(* Logix 5000 project; controller CarbonScout_MK6 vendor 1 type 14 code 154 rev 32.11; software revision 32.00; part 11 of 17 *)
(* tags used below, declared in another part *)
   ManualRunning : BOOL;
   ONS : BOOL[32];
   AI_FIT_01 : P_AIn;   // Purge water flow
   AI_LIT_01 : P_AIn;   // Carbon Scout Laser Level Transmitter
   AI_LIT_02 : P_AIn;   // Carbon Scout Cone Level Transmitter
   AI_PIT_01 : P_AIn;   // Water supply pressure
   AI_WIT_01 : P_AIn;   // Weight measure
   CS_Alarms : P_Alarm[80];
   CS_DINTParams : DINT[100];
   CS_REALParams : REAL[80];   // CS REAL Parameters
   CS_Result : CS_Results;   // Sample Result Live Async
   CS_Seq : GEK_Sequence;
   CS_Seq_ControlStop : BOOL;
   CS_Seq_CrashStop : BOOL;
   CS_Tank : CS_TankParams[20];
   CS_Timer : TIMER[80];
   CS_XRF : XRF;
   FOQ02 : TOTALIZER;   // Radar Calibration Totaliser
   N51 : DINT[5];   // From Client
   Oneshot : DINT;
   Oneshot2 : DINT;
   Oneshot3 : DINT;
   TimeAndDate : DINT[7];
   Valve_XV_01 : P_ValveSO;   // Sample Valve Tank 1
   Valve_XV_02 : P_ValveSO;   // Sample Valve Tank 2
   Valve_XV_03 : P_ValveSO;   // Sample Valve Tank 3
   Valve_XV_04 : P_ValveSO;   // Sample Valve Tank 4
   Valve_XV_05 : P_ValveSO;   // Sample Valve Tank 5
   Valve_XV_06 : P_ValveSO;   // Sample Valve Tank 6
   Valve_XV_07 : P_ValveSO;   // Sample Valve Tank 7
   Valve_XV_08 : P_ValveSO;   // Sample Valve Tank 8
   Valve_XV_09 : P_ValveSO;   // Sample Valve Tank 9
   Valve_XV_10 : P_ValveSO;   // Sample Valve Tank 10
   Valve_XV_11 : P_ValveSO;   // Purge Valve
   Valve_XV_12 : P_ValveSO;   // Slurry inlet vavle
   Valve_XV_13 : P_ValveSO;   // Sample line vavle
   Valve_XV_14 : P_ValveSO;   // Top wash vavle
   Valve_XV_15 : P_ValveSO;   // Bottme wash vavle
   Valve_XV_16 : P_ValveSO;   // Potable water valve / Supply Water Valve
   Valve_XV_17 : P_ValveSO;   // Sample cone outlet vavle
   Valve_XV_18 : P_ValveSO;   // Sample strainer discharge
   Valve_XV_19 : P_ValveSO;   // Laser window
(* SeqProgram, continued *)

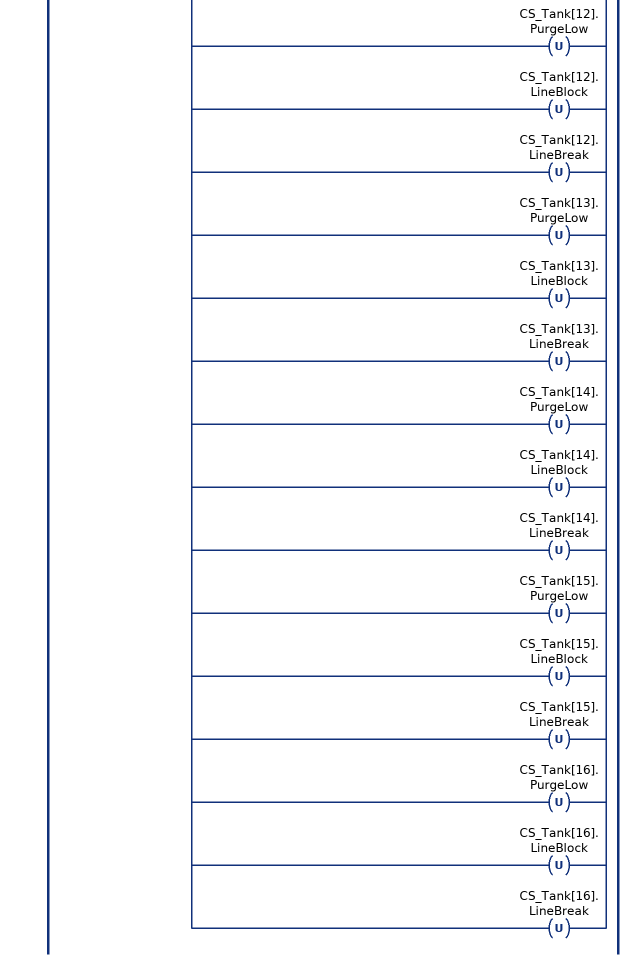
   83: XIC(CS_Seq.HMI_Reset_Req)[OTU(CS_Tank[1].PurgeLow) ,OTU(CS_Tank[1].LineBlock) ,OTU(CS_Tank[1].LineBreak) ,OTU(CS_Tank[2].PurgeLow) ,OTU(CS_Tank[2].LineBlock) ,OTU(CS_Tank[2].LineBreak) ,OTU(CS_Tank[3].PurgeLow) ,OTU(CS_Tank[3].LineBlock) ,OTU(CS_Tank[3].LineBreak) ,OTU(CS_Tank[4].PurgeLow) ,OTU(CS_Tank[4].LineBlock) ,OTU(CS_Tank[4].LineBreak) ,OTU(CS_Tank[5].PurgeLow) ,OTU(CS_Tank[5].LineBlock) ,OTU(CS_Tank[5].LineBreak) ,OTU(CS_Tank[6].PurgeLow) ,OTU(CS_Tank[6].LineBlock) ,OTU(CS_Tank[6].LineBreak) ,OTU(CS_Tank[7].PurgeLow) ,OTU(CS_Tank[7].LineBlock) ,OTU(CS_Tank[7].LineBreak) ,OTU(CS_Tank[8].PurgeLow) ,OTU(CS_Tank[8].LineBlock) ,OTU(CS_Tank[8].LineBreak) ,OTU(CS_Tank[9].PurgeLow) ,OTU(CS_Tank[9].LineBlock) ,OTU(CS_Tank[9].LineBreak) ,OTU(CS_Tank[10].PurgeLow) ,OTU(CS_Tank[10].LineBlock) ,OTU(CS_Tank[10].LineBreak) ,OTU(CS_Tank[11].PurgeLow) ,OTU(CS_Tank[11].LineBlock) ,OTU(CS_Tank[11].LineBreak) ,OTU(CS_Tank[12].PurgeLow) ,OTU(CS_Tank[12].LineBlock) ,OTU(CS_Tank[12].LineBreak) ,OTU(CS_Tank[13].PurgeLow) ,OTU(CS_Tank[13].LineBlock) ,OTU(CS_Tank[13].LineBreak) ,OTU(CS_Tank[14].PurgeLow) ,OTU(CS_Tank[14].LineBlock) ,OTU(CS_Tank[14].LineBreak) ,OTU(CS_Tank[15].PurgeLow) ,OTU(CS_Tank[15].LineBlock) ,OTU(CS_Tank[15].LineBreak) ,OTU(CS_Tank[16].PurgeLow) ,OTU(CS_Tank[16].LineBlock) ,OTU(CS_Tank[16].LineBreak) ];
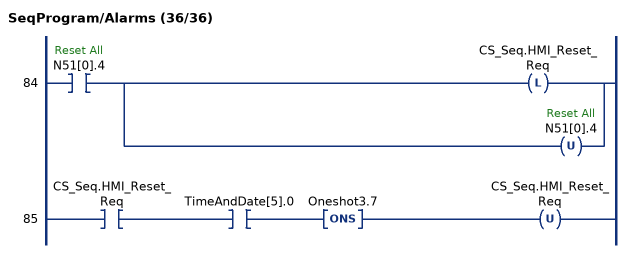
   84: XIC(N51[0].4)[OTL(CS_Seq.HMI_Reset_Req) ,OTU(N51[0].4) ];
   85: XIC(CS_Seq.HMI_Reset_Req)XIC(TimeAndDate[5].0)ONS(Oneshot3.7)OTU(CS_Seq.HMI_Reset_Req);
END_ROUTINE

ROUTINE AutoControl   (* ladder *)
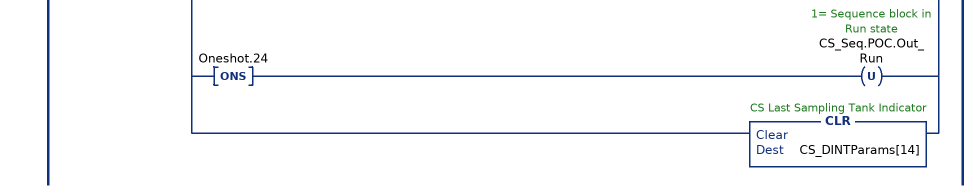
   // +++++++++++++++++++++++++++++
   // Gekko Batch/Continous Sequencer
   // Developed by TL and BT
   // +++++++++++++++++++++++++++++
   0: [MOV(0,CS_DINTParams[0]) P_Mode(CS_Seq.Mode) ,OTL(CS_Seq.Mode.Cfg_ProgDefault) ,DIV(CS_Seq.SeqTimer[0].ACC,1000,CS_DINTParams[1]) ,[XIC(CS_Seq.Mode.Sts_Prog) [[XIC(CS_Seq.HMI_Start_Req) ,XIC(CS_Timer[78].DN) ,XIC(N51[0].5) XIC(N51[0].0) ,XIC(CS_Seq.POC.Sts_Stopped) XIC(CS_DINTParams[99].11) [XIC(CS_DINTParams[97].0) XIC(CS_DINTParams[97].10) ,XIC(CS_DINTParams[97].1) XIC(CS_DINTParams[97].11) ,XIC(CS_DINTParams[97].2) XIC(CS_DINTParams[97].12) ,XIC(CS_DINTParams[97].3) XIC(CS_DINTParams[97].13) ,XIC(CS_DINTParams[97].4) XIC(CS_DINTParams[97].14) ,XIC(CS_DINTParams[97].5) XIC(CS_DINTParams[97].15) ,XIC(CS_DINTParams[97].6) XIC(CS_DINTParams[97].16) ,XIC(CS_DINTParams[97].7) XIC(CS_DINTParams[97].17) ,XIC(CS_DINTParams[97].8) XIC(CS_DINTParams[97].18) ,XIC(CS_DINTParams[97].9) XIC(CS_DINTParams[97].19) ] ] OTE(CS_Seq.POC.In_Cmd_Start) ,[XIC(CS_Seq.HMI_Pause_Req) ,LIM(1,N51[2],10) ] OTE(CS_Seq.POC.In_Cmd_Pause) ,[XIC(CS_Seq.HMI_StopPause_Req) ,XIC(N51[0].5) XIC(N51[0].1) ,LIM(11,N51[2],20) ] [AFI() OTE(CS_Seq.POC.In_Cmd_StopPause) ,OTL(CS_Seq_ControlStop) ] ] ,XIC(CS_Seq.Mode.Sts_Prog) [XIC(CS_Seq.HMI_Resume_Req) ,XIC(CS_Timer[78].DN) ] OTE(CS_Seq.POC.In_Cmd_Resume) ,XIC(CS_Seq.HMI_SkipF_Req) OTE(CS_Seq.POC.In_Cmd_SkipF) ,XIC(CS_Seq.HMI_SkipR_Req) OTE(CS_Seq.POC.In_Cmd_SkipR) ] ,OTL(CS_Seq.POC.In_Cfg_BatchContinous) MOV(23,CS_Seq.POC.In_MaxStepNum) MOV(2147483647,CS_Seq.SeqTimer[0].PRE) GekkoSeq(CS_Seq.POC,CS_Seq.SeqTimer[0]) ,[XIC(CS_Seq.POC.Sts_Running) ,XIC(CS_Seq.POC.Out_Run) ] [ONS(Oneshot.21) MOV(CS_Seq.POC.Out_MovingStepNum,CS_Seq.ActiveStage) ,MOV(CS_Seq.ActiveStage,CS_Seq.POC.In_StepNum) MOV(CS_Seq.ActiveStage,CS_Seq.POC.Out_MovingStepNum) ] ,XIC(CS_Seq.POC.Sts_Resumed) MOV(CS_Seq.POC.Out_NewStepNum,CS_Seq.ActiveStage) ,[XIO(CS_Seq.POC.Out_Run) XIO(CS_Seq.POC.Sts_StopPaused) XIO(CS_Seq.POC.Sts_Paused) XIO(CS_Seq.POC.Sts_Resumed) ,[[[XIC(CS_Seq_CrashStop) ,LIM(21,N51[2],30) ] ,XIC(S:FS) ] [CLR(CS_DINTParams[39]) ,OTU(CS_DINTParams[98].10) ] ,XIC(CS_Alarms[2].Alm) ] CLR(CS_Seq.POC.Out_MovingStepNum) ] MOV(0,CS_Seq.ActiveStage) ,EQU(CS_Seq.ActiveStage,0) OTE(CS_Seq.POC.In_Stopped) ,XIC(CS_Seq.POC.Out_Run) NEQ(CS_Seq.ActiveStage,0) OTE(CS_Seq.POC.In_Running) ,XIC(CS_Seq.POC.Sts_Stopped) [XIC(CS_Seq.POC.Sts_Paused) OTU(CS_Seq.POC.Sts_Paused) ,XIC(CS_Seq.POC.Sts_StopPaused) OTU(CS_Seq.POC.Sts_StopPaused) ,OTU(CS_Seq_ControlStop) ,OTU(CS_DINTParams[99].23) ,OTU(CS_DINTParams[99].10) ,OTU(CS_DINTParams[99].7) MOV(0,CS_Result.ErrorFlag) ,OTU(CS_DINTParams[99].8) ,ONS(Oneshot.24) OTU(CS_Seq.POC.Out_Run) ,CLR(CS_DINTParams[14]) ] ];
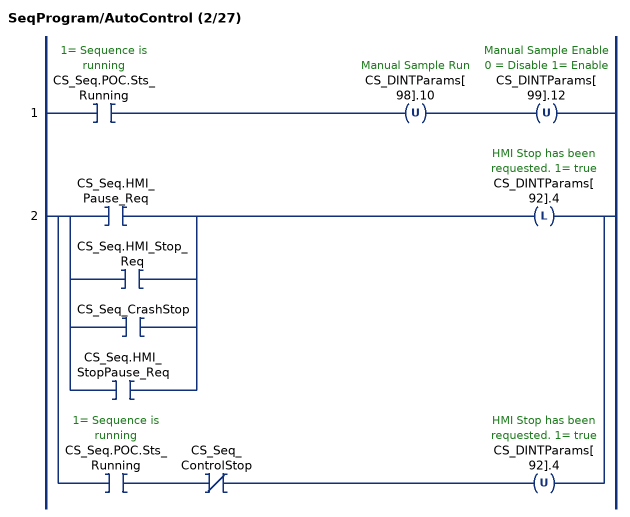
   1: XIC(CS_Seq.POC.Sts_Running)OTU(CS_DINTParams[98].10)OTU(CS_DINTParams[99].12);
   2: [[XIC(CS_Seq.HMI_Pause_Req) ,XIC(CS_Seq.HMI_Stop_Req) ,XIC(CS_Seq_CrashStop) ,XIC(CS_Seq.HMI_StopPause_Req) ] OTL(CS_DINTParams[92].4) ,XIC(CS_Seq.POC.Sts_Running) XIO(CS_Seq_ControlStop) OTU(CS_DINTParams[92].4) ];
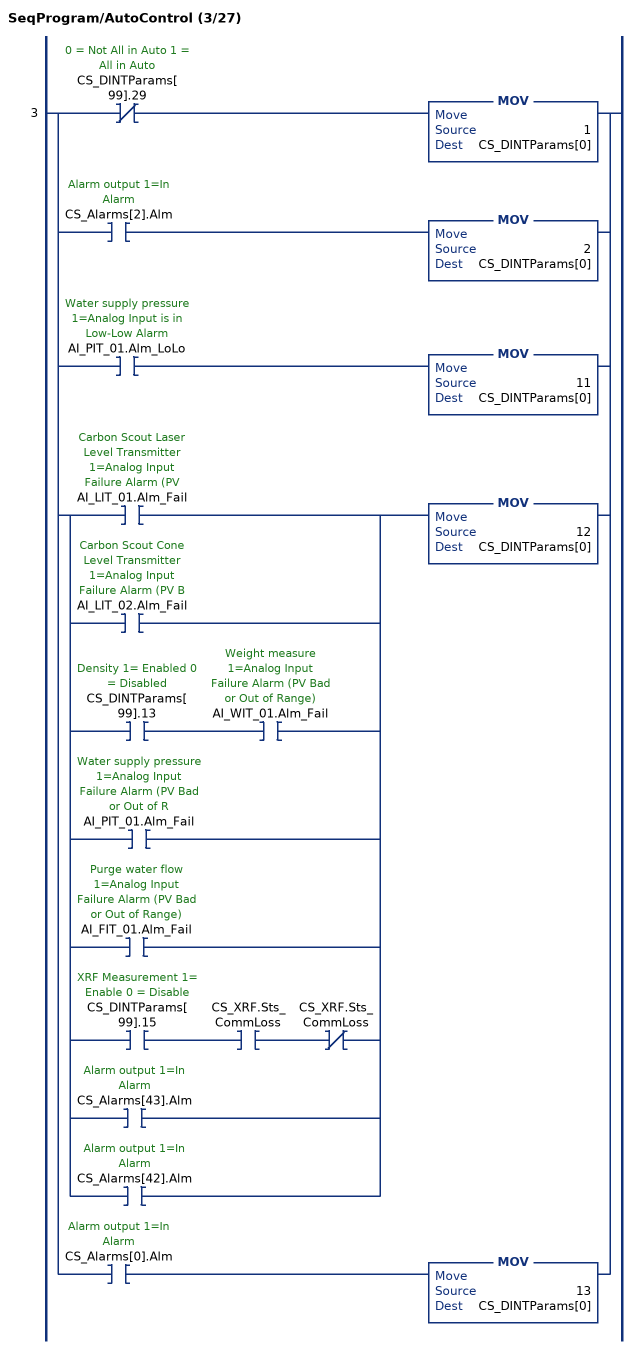
   3: [XIO(CS_DINTParams[99].29) MOV(1,CS_DINTParams[0]) ,XIC(CS_Alarms[2].Alm) MOV(2,CS_DINTParams[0]) ,XIC(AI_PIT_01.Alm_LoLo) MOV(11,CS_DINTParams[0]) ,[XIC(AI_LIT_01.Alm_Fail) ,XIC(AI_LIT_02.Alm_Fail) ,XIC(CS_DINTParams[99].13) XIC(AI_WIT_01.Alm_Fail) ,XIC(AI_PIT_01.Alm_Fail) ,XIC(AI_FIT_01.Alm_Fail) ,XIC(CS_DINTParams[99].15) XIC(CS_XRF.Sts_CommLoss) XIO(CS_XRF.Sts_CommLoss) ,XIC(CS_Alarms[43].Alm) ,XIC(CS_Alarms[42].Alm) ] MOV(12,CS_DINTParams[0]) ,XIC(CS_Alarms[0].Alm) MOV(13,CS_DINTParams[0]) ];
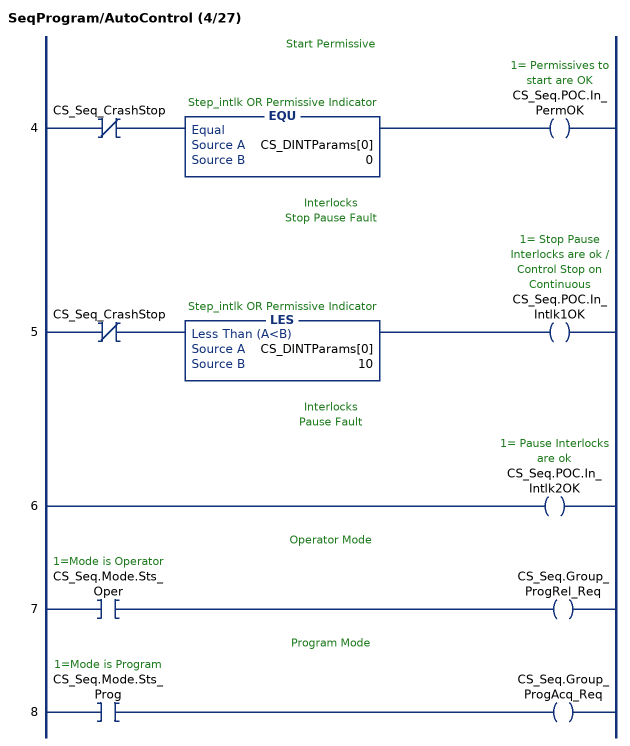
   // Start Permissive
   4: XIO(CS_Seq_CrashStop)EQU(CS_DINTParams[0],0)OTE(CS_Seq.POC.In_PermOK);
   // Interlocks
   // Stop Pause Fault
   5: XIO(CS_Seq_CrashStop)LES(CS_DINTParams[0],10)OTE(CS_Seq.POC.In_Intlk1OK);
   // Interlocks
   // Pause Fault
   6: OTE(CS_Seq.POC.In_Intlk2OK);
   // Operator Mode
   7: XIC(CS_Seq.Mode.Sts_Oper)OTE(CS_Seq.Group_ProgRel_Req);
   // Program Mode
   8: XIC(CS_Seq.Mode.Sts_Prog)OTE(CS_Seq.Group_ProgAcq_Req);
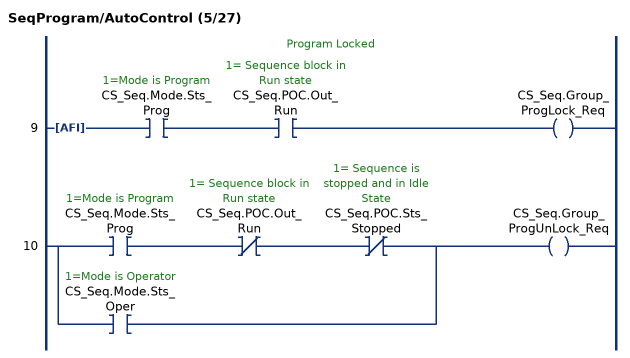
   // Program Locked
   9: AFI()XIC(CS_Seq.Mode.Sts_Prog)XIC(CS_Seq.POC.Out_Run)OTE(CS_Seq.Group_ProgLock_Req);
   10: [XIC(CS_Seq.Mode.Sts_Prog) XIO(CS_Seq.POC.Out_Run) XIO(CS_Seq.POC.Sts_Stopped) ,XIC(CS_Seq.Mode.Sts_Oper) ]OTE(CS_Seq.Group_ProgUnLock_Req);
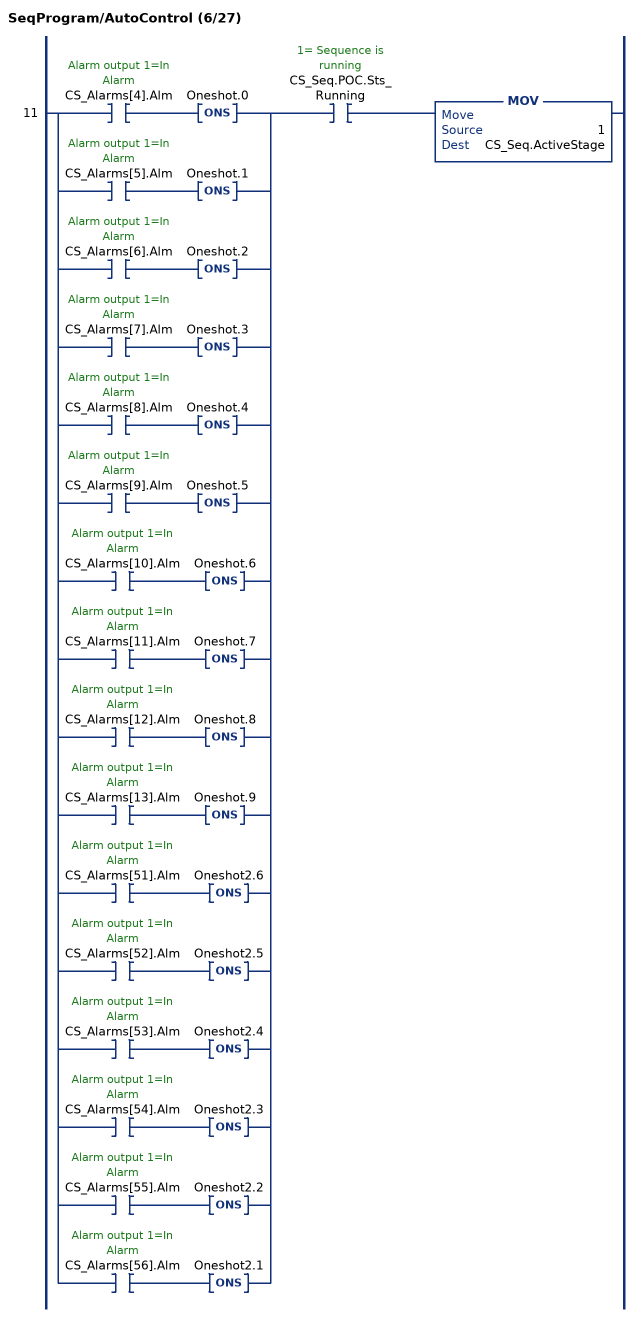
   11: [XIC(CS_Alarms[4].Alm) ONS(Oneshot.0) ,XIC(CS_Alarms[5].Alm) ONS(Oneshot.1) ,XIC(CS_Alarms[6].Alm) ONS(Oneshot.2) ,XIC(CS_Alarms[7].Alm) ONS(Oneshot.3) ,XIC(CS_Alarms[8].Alm) ONS(Oneshot.4) ,XIC(CS_Alarms[9].Alm) ONS(Oneshot.5) ,XIC(CS_Alarms[10].Alm) ONS(Oneshot.6) ,XIC(CS_Alarms[11].Alm) ONS(Oneshot.7) ,XIC(CS_Alarms[12].Alm) ONS(Oneshot.8) ,XIC(CS_Alarms[13].Alm) ONS(Oneshot.9) ,XIC(CS_Alarms[51].Alm) ONS(Oneshot2.6) ,XIC(CS_Alarms[52].Alm) ONS(Oneshot2.5) ,XIC(CS_Alarms[53].Alm) ONS(Oneshot2.4) ,XIC(CS_Alarms[54].Alm) ONS(Oneshot2.3) ,XIC(CS_Alarms[55].Alm) ONS(Oneshot2.2) ,XIC(CS_Alarms[56].Alm) ONS(Oneshot2.1) ]XIC(CS_Seq.POC.Sts_Running)MOV(1,CS_Seq.ActiveStage);
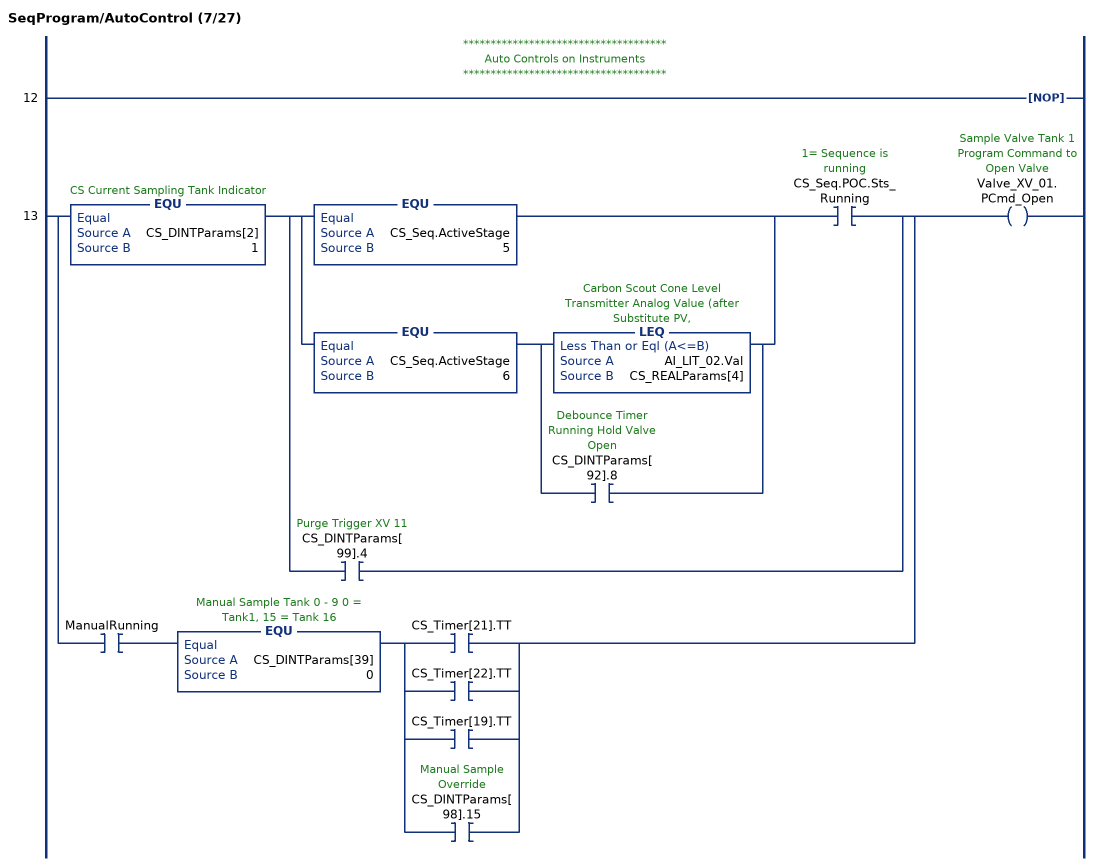
   // *************************************
   // Auto Controls on Instruments
   // *************************************
   12: NOP();
   13: [EQU(CS_DINTParams[2],1) [[EQU(CS_Seq.ActiveStage,5) ,EQU(CS_Seq.ActiveStage,6) [LEQ(AI_LIT_02.Val,CS_REALParams[4]) ,XIC(CS_DINTParams[92].8) ] ] XIC(CS_Seq.POC.Sts_Running) ,XIC(CS_DINTParams[99].4) ] ,XIC(ManualRunning) EQU(CS_DINTParams[39],0) [XIC(CS_Timer[21].TT) ,XIC(CS_Timer[22].TT) ,XIC(CS_Timer[19].TT) ,XIC(CS_DINTParams[98].15) ] ]OTE(Valve_XV_01.PCmd_Open);
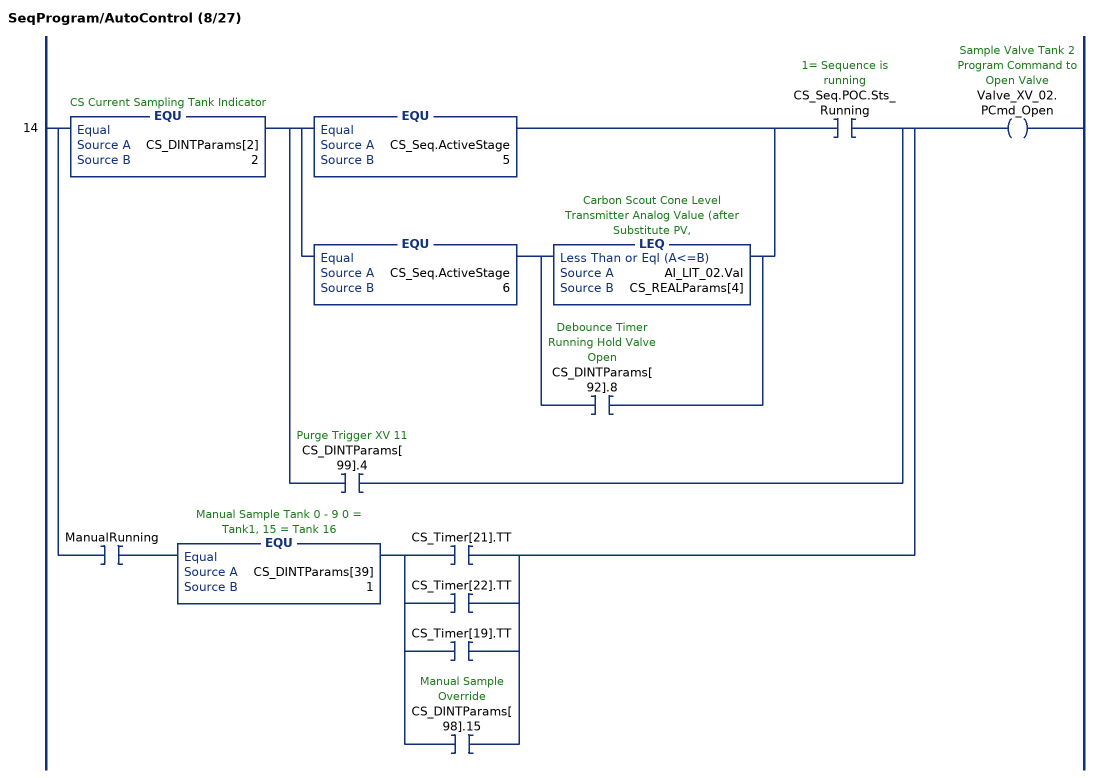
   14: [EQU(CS_DINTParams[2],2) [[EQU(CS_Seq.ActiveStage,5) ,EQU(CS_Seq.ActiveStage,6) [LEQ(AI_LIT_02.Val,CS_REALParams[4]) ,XIC(CS_DINTParams[92].8) ] ] XIC(CS_Seq.POC.Sts_Running) ,XIC(CS_DINTParams[99].4) ] ,XIC(ManualRunning) EQU(CS_DINTParams[39],1) [XIC(CS_Timer[21].TT) ,XIC(CS_Timer[22].TT) ,XIC(CS_Timer[19].TT) ,XIC(CS_DINTParams[98].15) ] ]OTE(Valve_XV_02.PCmd_Open);
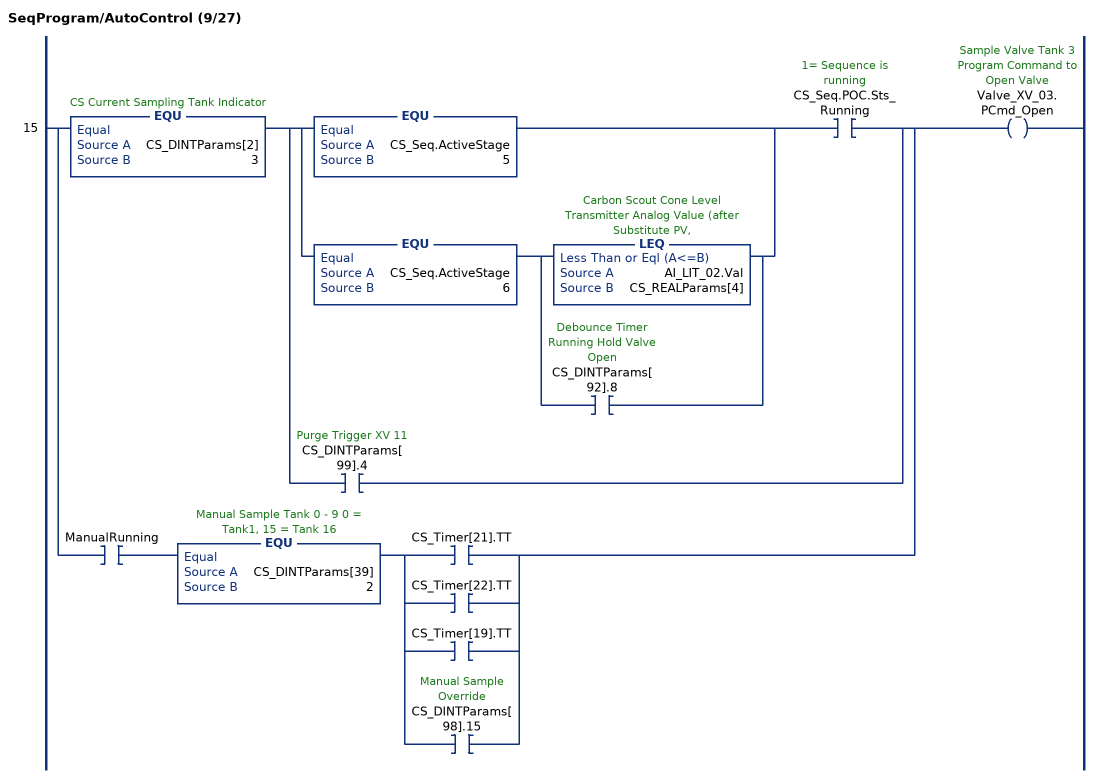
   15: [EQU(CS_DINTParams[2],3) [[EQU(CS_Seq.ActiveStage,5) ,EQU(CS_Seq.ActiveStage,6) [LEQ(AI_LIT_02.Val,CS_REALParams[4]) ,XIC(CS_DINTParams[92].8) ] ] XIC(CS_Seq.POC.Sts_Running) ,XIC(CS_DINTParams[99].4) ] ,XIC(ManualRunning) EQU(CS_DINTParams[39],2) [XIC(CS_Timer[21].TT) ,XIC(CS_Timer[22].TT) ,XIC(CS_Timer[19].TT) ,XIC(CS_DINTParams[98].15) ] ]OTE(Valve_XV_03.PCmd_Open);
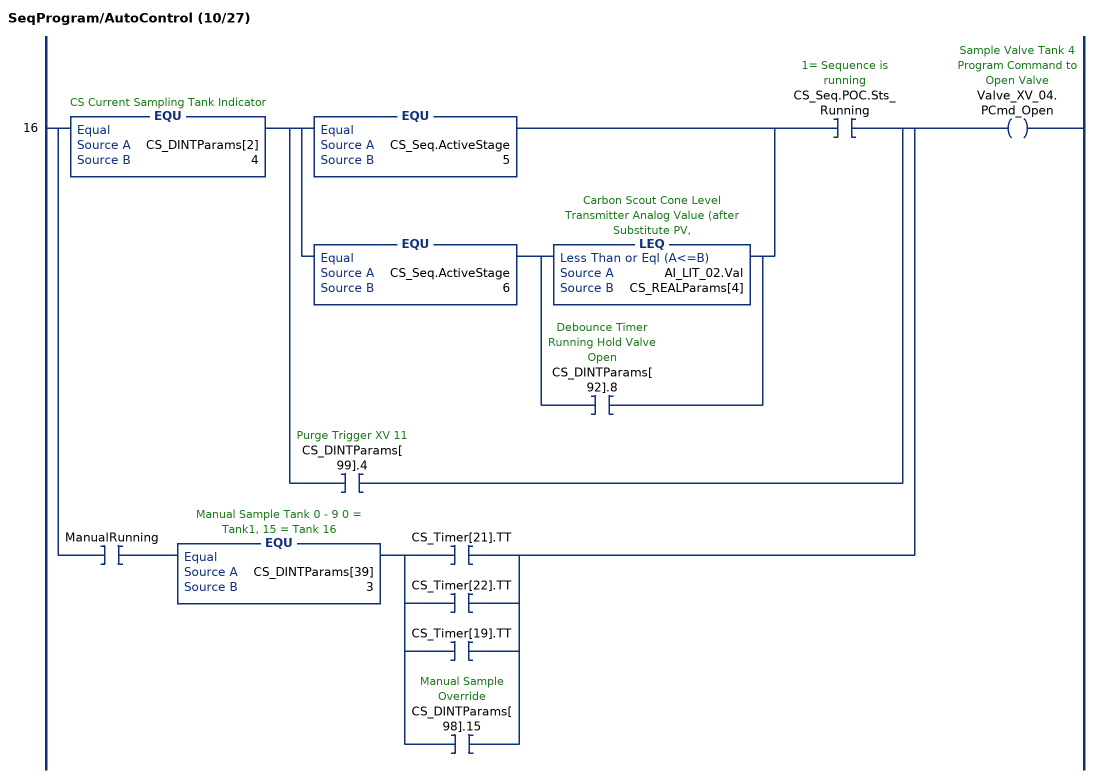
   16: [EQU(CS_DINTParams[2],4) [[EQU(CS_Seq.ActiveStage,5) ,EQU(CS_Seq.ActiveStage,6) [LEQ(AI_LIT_02.Val,CS_REALParams[4]) ,XIC(CS_DINTParams[92].8) ] ] XIC(CS_Seq.POC.Sts_Running) ,XIC(CS_DINTParams[99].4) ] ,XIC(ManualRunning) EQU(CS_DINTParams[39],3) [XIC(CS_Timer[21].TT) ,XIC(CS_Timer[22].TT) ,XIC(CS_Timer[19].TT) ,XIC(CS_DINTParams[98].15) ] ]OTE(Valve_XV_04.PCmd_Open);
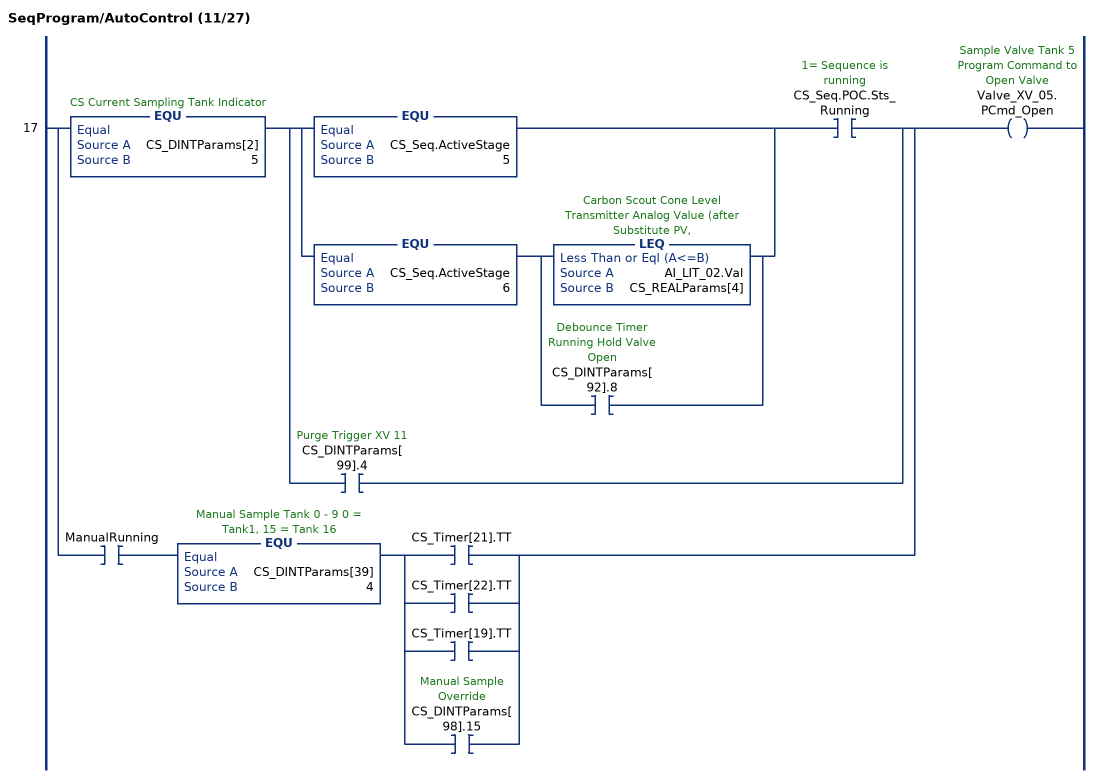
   17: [EQU(CS_DINTParams[2],5) [[EQU(CS_Seq.ActiveStage,5) ,EQU(CS_Seq.ActiveStage,6) [LEQ(AI_LIT_02.Val,CS_REALParams[4]) ,XIC(CS_DINTParams[92].8) ] ] XIC(CS_Seq.POC.Sts_Running) ,XIC(CS_DINTParams[99].4) ] ,XIC(ManualRunning) EQU(CS_DINTParams[39],4) [XIC(CS_Timer[21].TT) ,XIC(CS_Timer[22].TT) ,XIC(CS_Timer[19].TT) ,XIC(CS_DINTParams[98].15) ] ]OTE(Valve_XV_05.PCmd_Open);
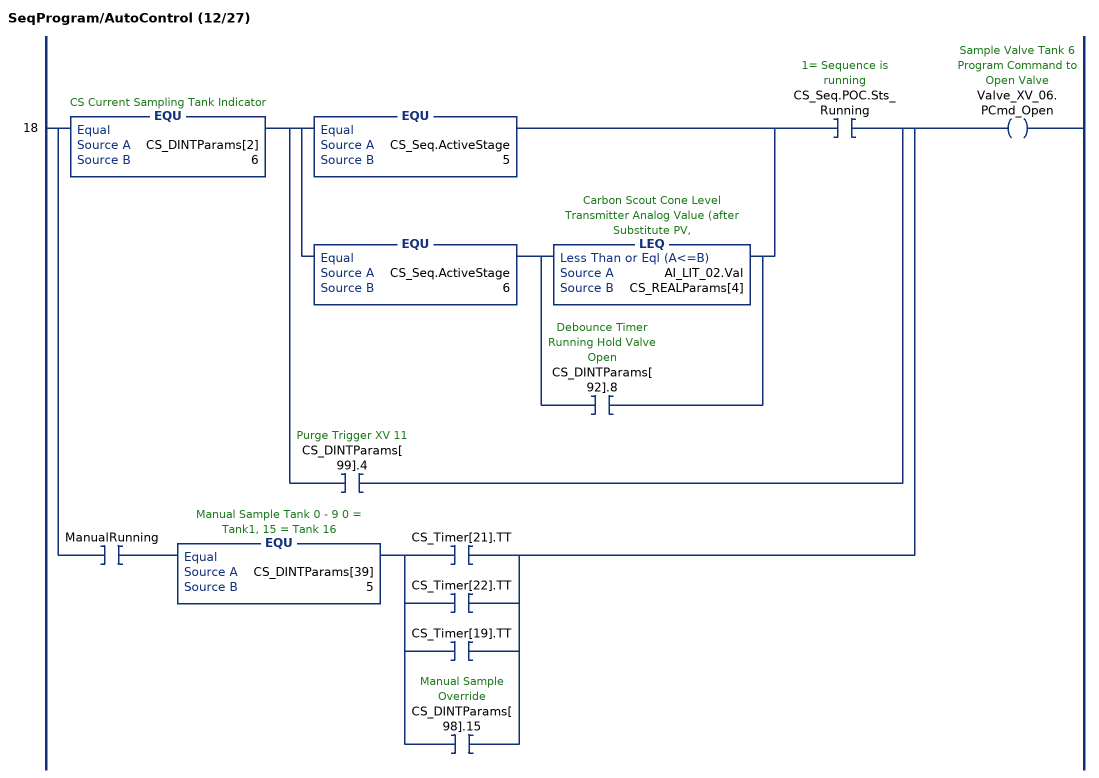
   18: [EQU(CS_DINTParams[2],6) [[EQU(CS_Seq.ActiveStage,5) ,EQU(CS_Seq.ActiveStage,6) [LEQ(AI_LIT_02.Val,CS_REALParams[4]) ,XIC(CS_DINTParams[92].8) ] ] XIC(CS_Seq.POC.Sts_Running) ,XIC(CS_DINTParams[99].4) ] ,XIC(ManualRunning) EQU(CS_DINTParams[39],5) [XIC(CS_Timer[21].TT) ,XIC(CS_Timer[22].TT) ,XIC(CS_Timer[19].TT) ,XIC(CS_DINTParams[98].15) ] ]OTE(Valve_XV_06.PCmd_Open);
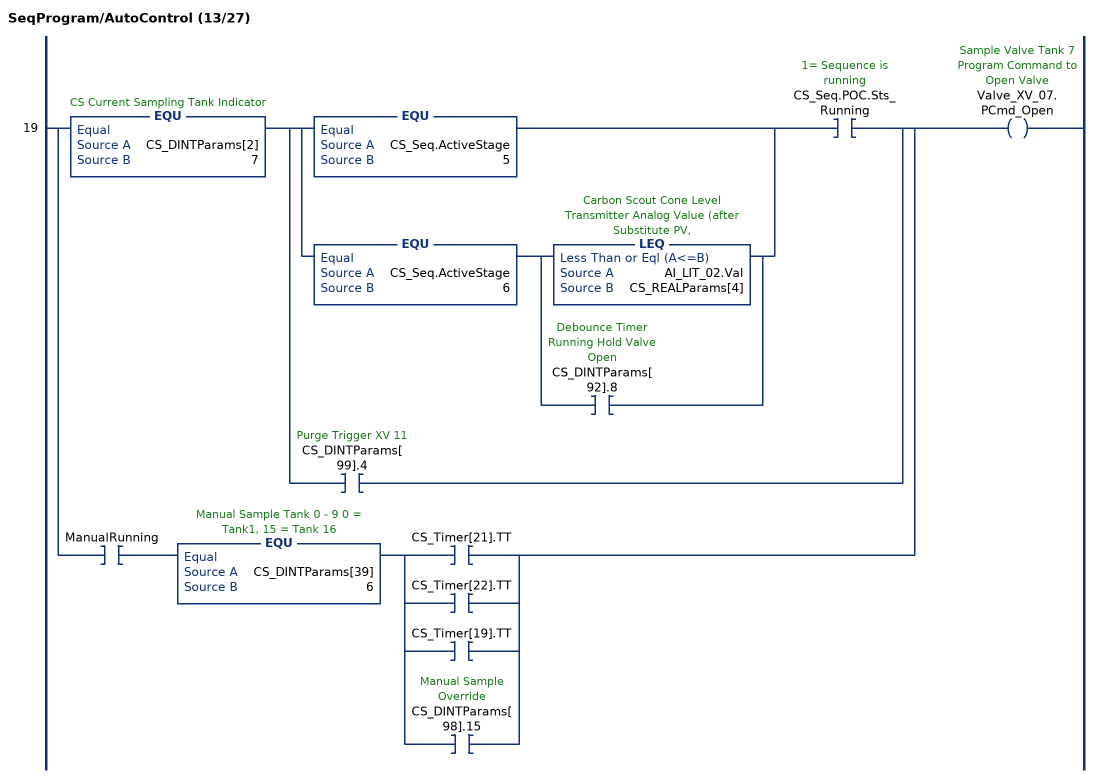
   19: [EQU(CS_DINTParams[2],7) [[EQU(CS_Seq.ActiveStage,5) ,EQU(CS_Seq.ActiveStage,6) [LEQ(AI_LIT_02.Val,CS_REALParams[4]) ,XIC(CS_DINTParams[92].8) ] ] XIC(CS_Seq.POC.Sts_Running) ,XIC(CS_DINTParams[99].4) ] ,XIC(ManualRunning) EQU(CS_DINTParams[39],6) [XIC(CS_Timer[21].TT) ,XIC(CS_Timer[22].TT) ,XIC(CS_Timer[19].TT) ,XIC(CS_DINTParams[98].15) ] ]OTE(Valve_XV_07.PCmd_Open);
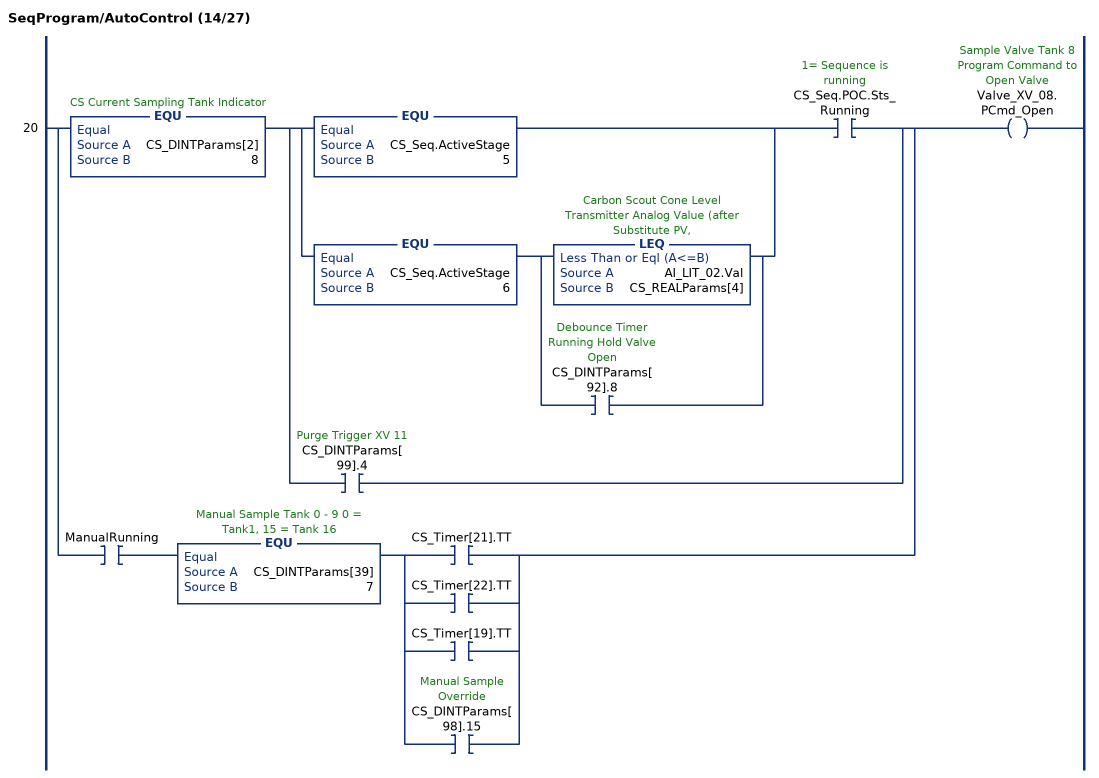
   20: [EQU(CS_DINTParams[2],8) [[EQU(CS_Seq.ActiveStage,5) ,EQU(CS_Seq.ActiveStage,6) [LEQ(AI_LIT_02.Val,CS_REALParams[4]) ,XIC(CS_DINTParams[92].8) ] ] XIC(CS_Seq.POC.Sts_Running) ,XIC(CS_DINTParams[99].4) ] ,XIC(ManualRunning) EQU(CS_DINTParams[39],7) [XIC(CS_Timer[21].TT) ,XIC(CS_Timer[22].TT) ,XIC(CS_Timer[19].TT) ,XIC(CS_DINTParams[98].15) ] ]OTE(Valve_XV_08.PCmd_Open);
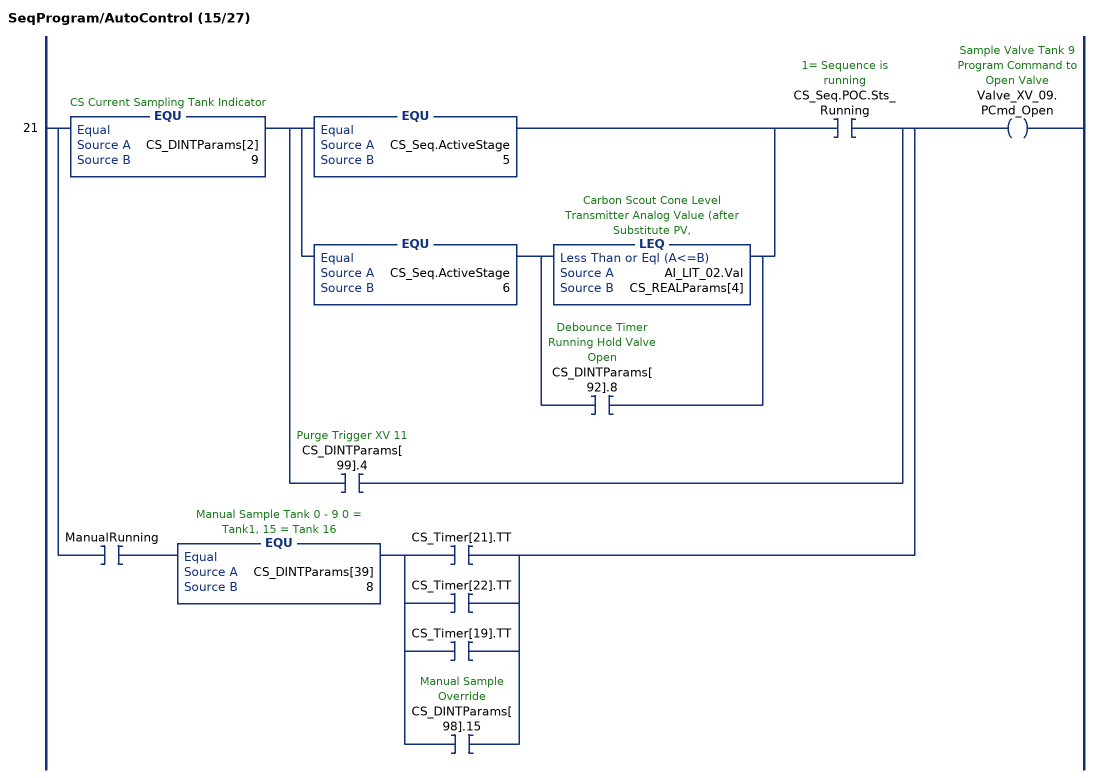
   21: [EQU(CS_DINTParams[2],9) [[EQU(CS_Seq.ActiveStage,5) ,EQU(CS_Seq.ActiveStage,6) [LEQ(AI_LIT_02.Val,CS_REALParams[4]) ,XIC(CS_DINTParams[92].8) ] ] XIC(CS_Seq.POC.Sts_Running) ,XIC(CS_DINTParams[99].4) ] ,XIC(ManualRunning) EQU(CS_DINTParams[39],8) [XIC(CS_Timer[21].TT) ,XIC(CS_Timer[22].TT) ,XIC(CS_Timer[19].TT) ,XIC(CS_DINTParams[98].15) ] ]OTE(Valve_XV_09.PCmd_Open);
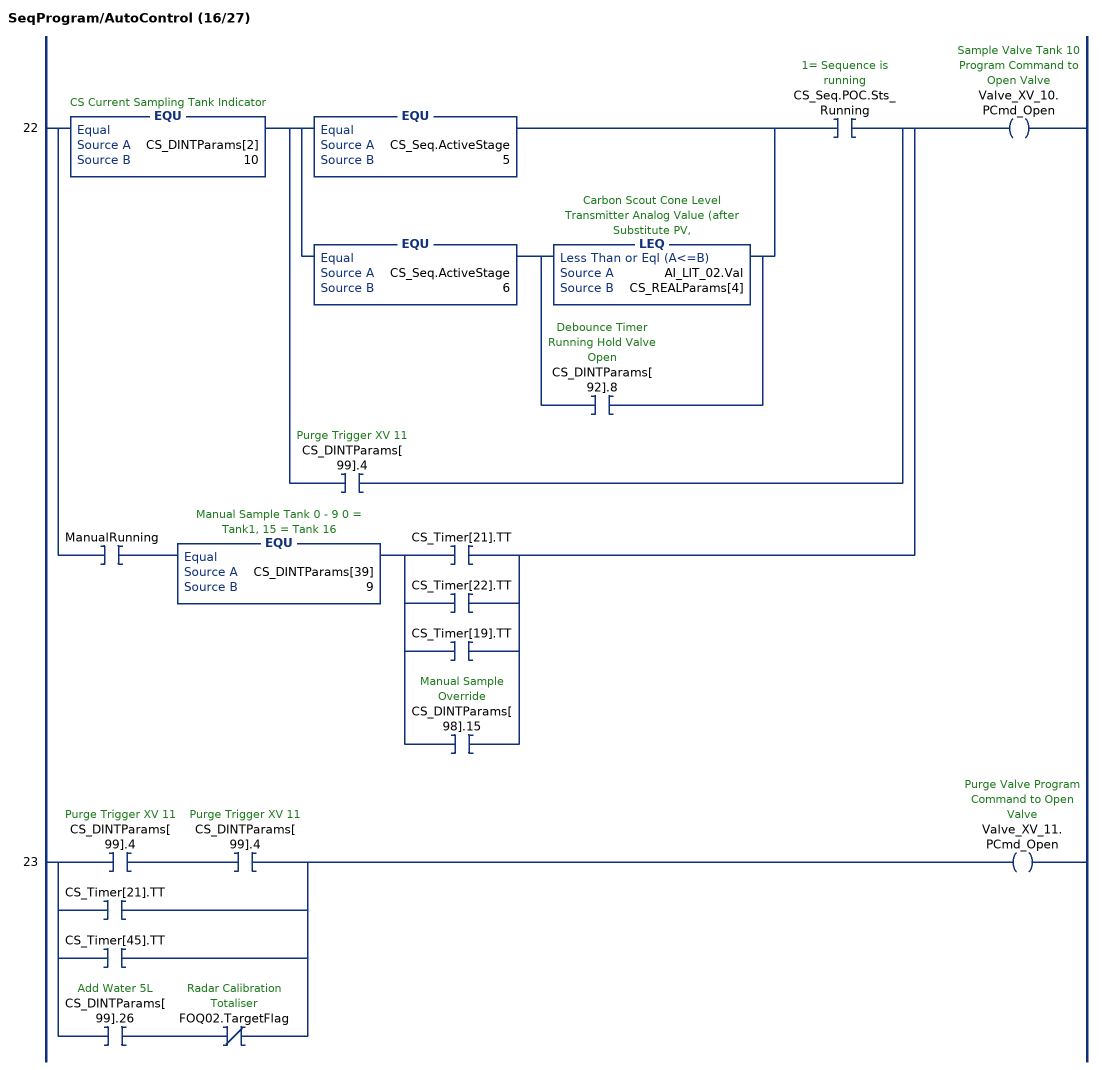
   22: [EQU(CS_DINTParams[2],10) [[EQU(CS_Seq.ActiveStage,5) ,EQU(CS_Seq.ActiveStage,6) [LEQ(AI_LIT_02.Val,CS_REALParams[4]) ,XIC(CS_DINTParams[92].8) ] ] XIC(CS_Seq.POC.Sts_Running) ,XIC(CS_DINTParams[99].4) ] ,XIC(ManualRunning) EQU(CS_DINTParams[39],9) [XIC(CS_Timer[21].TT) ,XIC(CS_Timer[22].TT) ,XIC(CS_Timer[19].TT) ,XIC(CS_DINTParams[98].15) ] ]OTE(Valve_XV_10.PCmd_Open);
   23: [XIC(CS_DINTParams[99].4) XIC(CS_DINTParams[99].4) ,XIC(CS_Timer[21].TT) ,XIC(CS_Timer[45].TT) ,XIC(CS_DINTParams[99].26) XIO(FOQ02.TargetFlag) ]OTE(Valve_XV_11.PCmd_Open);
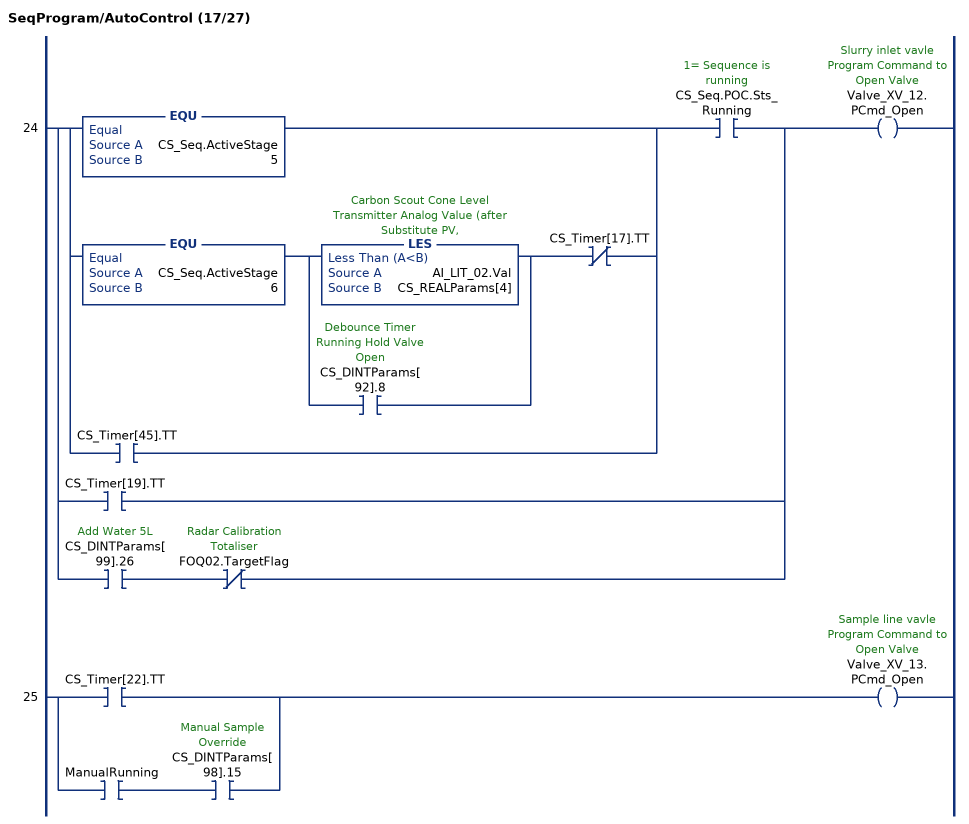
   24: [[EQU(CS_Seq.ActiveStage,5) ,EQU(CS_Seq.ActiveStage,6) [LES(AI_LIT_02.Val,CS_REALParams[4]) ,XIC(CS_DINTParams[92].8) ] XIO(CS_Timer[17].TT) ,XIC(CS_Timer[45].TT) ] XIC(CS_Seq.POC.Sts_Running) ,XIC(CS_Timer[19].TT) ,XIC(CS_DINTParams[99].26) XIO(FOQ02.TargetFlag) ]OTE(Valve_XV_12.PCmd_Open);
   25: [XIC(CS_Timer[22].TT) ,XIC(ManualRunning) XIC(CS_DINTParams[98].15) ]OTE(Valve_XV_13.PCmd_Open);
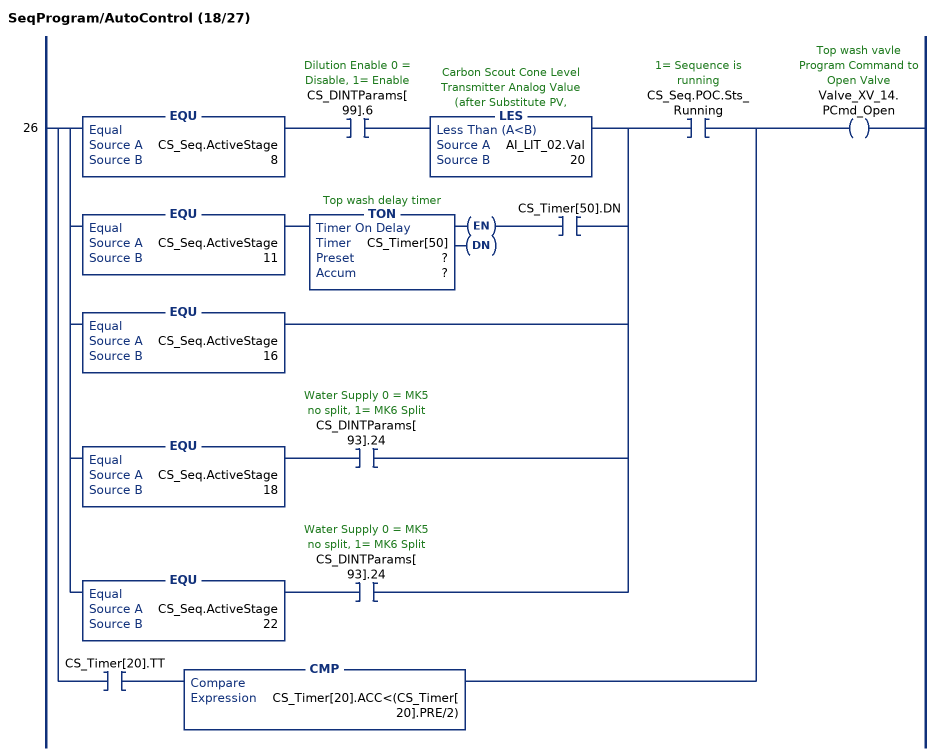
   26: [[EQU(CS_Seq.ActiveStage,8) XIC(CS_DINTParams[99].6) LES(AI_LIT_02.Val,20) ,EQU(CS_Seq.ActiveStage,11) TON(CS_Timer[50],?,?) XIC(CS_Timer[50].DN) ,EQU(CS_Seq.ActiveStage,16) ,EQU(CS_Seq.ActiveStage,18) XIC(CS_DINTParams[93].24) ,EQU(CS_Seq.ActiveStage,22) XIC(CS_DINTParams[93].24) ] XIC(CS_Seq.POC.Sts_Running) ,XIC(CS_Timer[20].TT) CMP(CS_Timer[20].ACC<(CS_Timer[20].PRE/2)) ]OTE(Valve_XV_14.PCmd_Open);
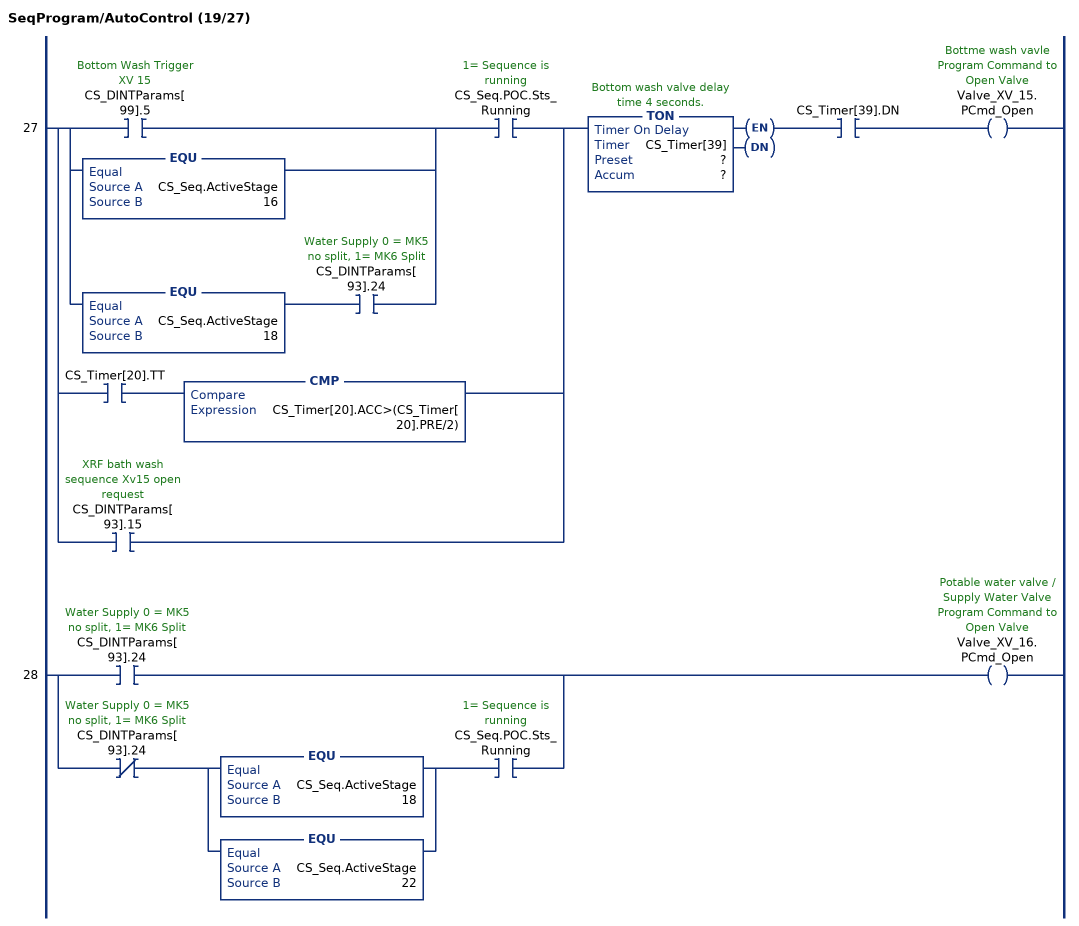
   27: [[XIC(CS_DINTParams[99].5) ,EQU(CS_Seq.ActiveStage,16) ,EQU(CS_Seq.ActiveStage,18) XIC(CS_DINTParams[93].24) ] XIC(CS_Seq.POC.Sts_Running) ,XIC(CS_Timer[20].TT) CMP(CS_Timer[20].ACC>(CS_Timer[20].PRE/2)) ,XIC(CS_DINTParams[93].15) ]TON(CS_Timer[39],?,?)XIC(CS_Timer[39].DN)OTE(Valve_XV_15.PCmd_Open);
   28: [XIC(CS_DINTParams[93].24) ,XIO(CS_DINTParams[93].24) [EQU(CS_Seq.ActiveStage,18) ,EQU(CS_Seq.ActiveStage,22) ] XIC(CS_Seq.POC.Sts_Running) ]OTE(Valve_XV_16.PCmd_Open);
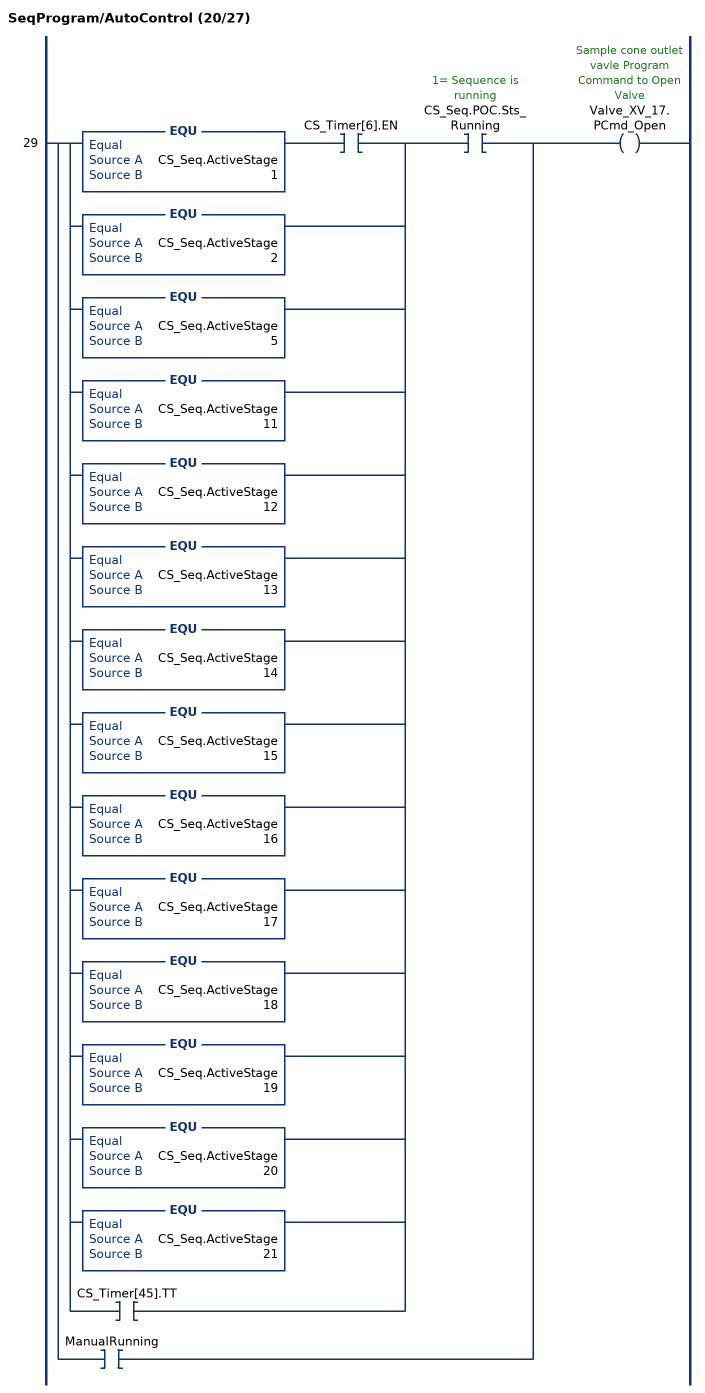
   29: [[EQU(CS_Seq.ActiveStage,1) XIC(CS_Timer[6].EN) ,EQU(CS_Seq.ActiveStage,2) ,EQU(CS_Seq.ActiveStage,5) ,EQU(CS_Seq.ActiveStage,11) ,EQU(CS_Seq.ActiveStage,12) ,EQU(CS_Seq.ActiveStage,13) ,EQU(CS_Seq.ActiveStage,14) ,EQU(CS_Seq.ActiveStage,15) ,EQU(CS_Seq.ActiveStage,16) ,EQU(CS_Seq.ActiveStage,17) ,EQU(CS_Seq.ActiveStage,18) ,EQU(CS_Seq.ActiveStage,19) ,EQU(CS_Seq.ActiveStage,20) ,EQU(CS_Seq.ActiveStage,21) ,XIC(CS_Timer[45].TT) ] XIC(CS_Seq.POC.Sts_Running) ,XIC(ManualRunning) ]OTE(Valve_XV_17.PCmd_Open);
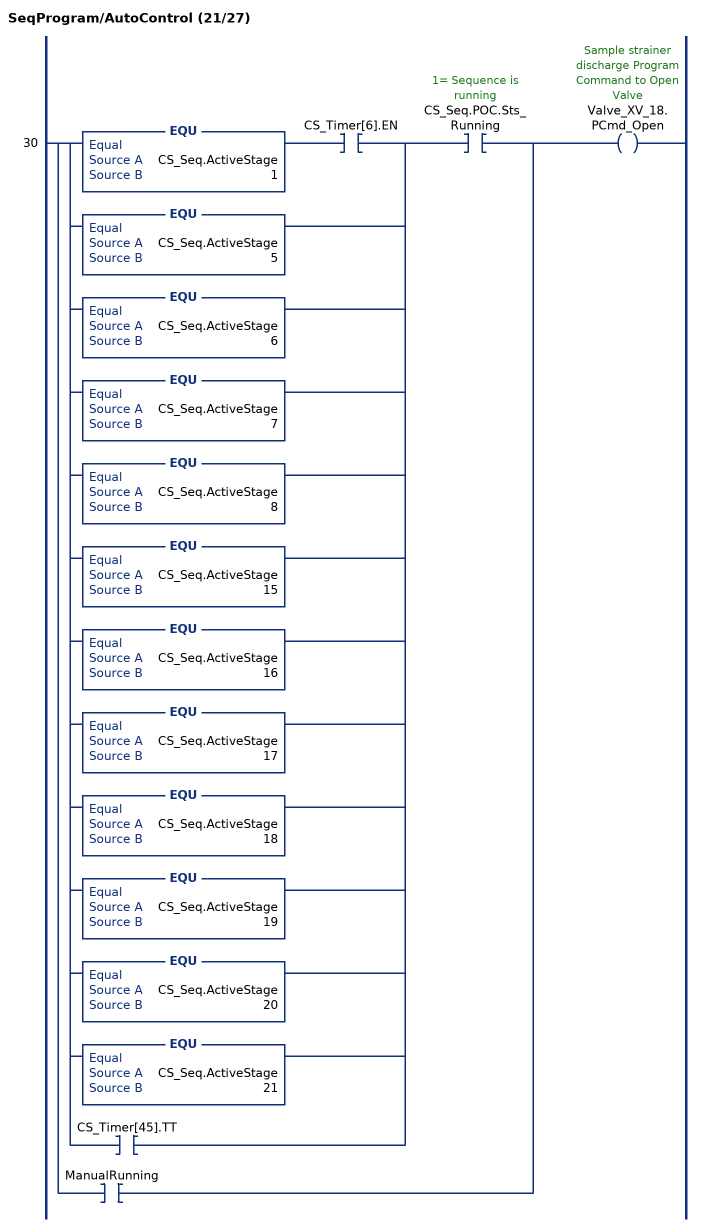
   30: [[EQU(CS_Seq.ActiveStage,1) XIC(CS_Timer[6].EN) ,EQU(CS_Seq.ActiveStage,5) ,EQU(CS_Seq.ActiveStage,6) ,EQU(CS_Seq.ActiveStage,7) ,EQU(CS_Seq.ActiveStage,8) ,EQU(CS_Seq.ActiveStage,15) ,EQU(CS_Seq.ActiveStage,16) ,EQU(CS_Seq.ActiveStage,17) ,EQU(CS_Seq.ActiveStage,18) ,EQU(CS_Seq.ActiveStage,19) ,EQU(CS_Seq.ActiveStage,20) ,EQU(CS_Seq.ActiveStage,21) ,XIC(CS_Timer[45].TT) ] XIC(CS_Seq.POC.Sts_Running) ,XIC(ManualRunning) ]OTE(Valve_XV_18.PCmd_Open);
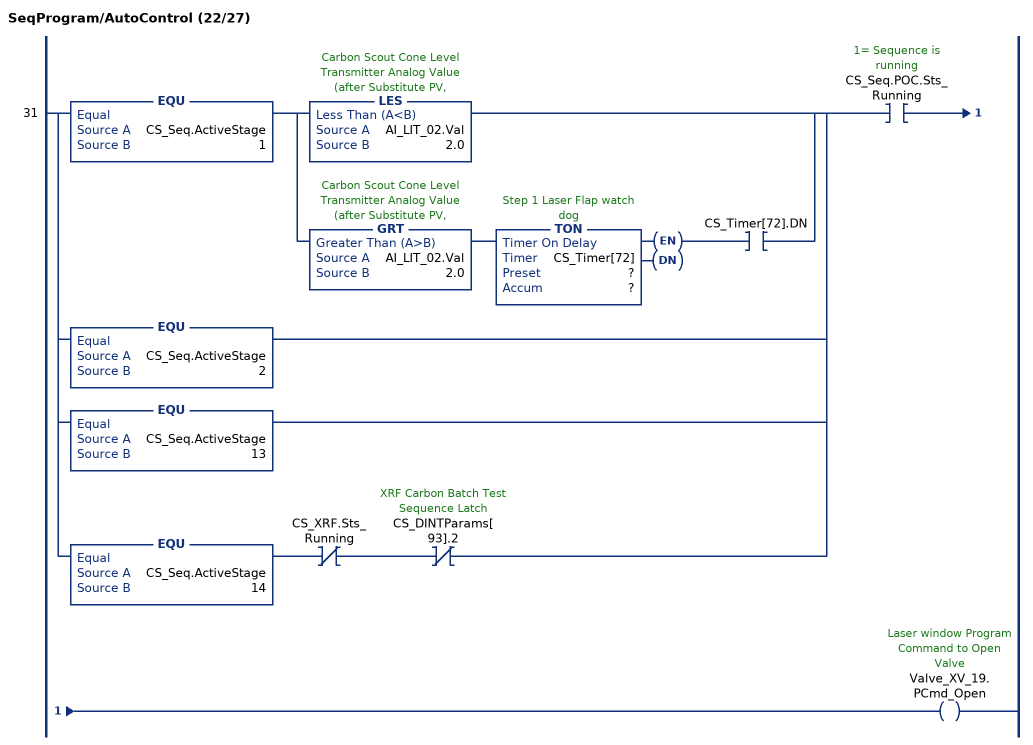
   31: [EQU(CS_Seq.ActiveStage,1) [LES(AI_LIT_02.Val,2.0) ,GRT(AI_LIT_02.Val,2.0) TON(CS_Timer[72],?,?) XIC(CS_Timer[72].DN) ] ,EQU(CS_Seq.ActiveStage,2) ,EQU(CS_Seq.ActiveStage,13) ,EQU(CS_Seq.ActiveStage,14) XIO(CS_XRF.Sts_Running) XIO(CS_DINTParams[93].2) ]XIC(CS_Seq.POC.Sts_Running)OTE(Valve_XV_19.PCmd_Open);
